Staubli VAL3: OnF4.pgx

public program OnF4()
begin
end
